TYPE Safety_Zones :
STRUCT
	Front_back_white_zone : BOOL := FALSE ;
	Front_back_red_zone : BOOL := FALSE ;
	Front_back_purple_zone : BOOL := TRUE ;
	Front_back_grey_pink_zone : BOOL := TRUE ;
	
END_STRUCT
END_TYPE

(* stored: Version 1.1.0.1, ProductVersion 3.1.4024.12
   DUT Safety_Zones: Id {b0881910-44f7-4580-abc0-e21e14826f5f} *)
